TYPE ST_Event :
STRUCT
	eEventType : E_EventType;
	eEventSeverity : TcEventSeverity;
	nEventIdentity : E_EventIDs;
	sSourceName : STRING(255);
	sEventText : STRING(255);
	dtTimestamp : DATE_AND_TIME;
	eTimeZoneID : E_TimeZoneID;
END_STRUCT
END_TYPE

(* stored: Version 1.1.0.1, ProductVersion 3.1.4024.11
   DUT ST_Event: Id {4e2b668f-cc82-4568-b54e-0d5da6f117b3} *)
